  MoveL 730 to (129.65, 249.05, 0) mm, rotated rx 180 ry 0 rz -39.83 deg; joints [47.121, -60.596, 63.822, -0.862, 86.762, 47.166]
  MoveL 731 to (129.42, 249.1, 0) mm, rotated rx -180 ry 0 rz -39.83 deg; joints [47.111, -60.591, 63.814, -0.862, 86.764, 47.156]
  MoveL 732 to (129.2, 249.14, 0) mm, rotated rx -180 ry 0 rz -39.83 deg; joints [47.101, -60.586, 63.806, -0.862, 86.767, 47.146]
  MoveL 733 to (128.97, 249.18, 0) mm, rotated rx 180 ry 0 rz -39.83 deg; joints [47.091, -60.582, 63.799, -0.862, 86.769, 47.136]
  MoveL 734 to (128.75, 249.21, 0) mm, rotated rx 180 ry 0 rz -39.83 deg; joints [47.081, -60.577, 63.792, -0.862, 86.772, 47.126]
  MoveL 735 to (128.47, 249.26, 0) mm, rotated rx -180 ry 0 rz -39.83 deg; joints [47.068, -60.572, 63.784, -0.862, 86.775, 47.113]
  MoveL 736 to (128.19, 249.3, 0) mm, rotated rx 180 ry 0 rz -39.83 deg; joints [47.056, -60.567, 63.776, -0.862, 86.777, 47.101]
  MoveL 737 to (127.92, 249.33, 0) mm, rotated rx 180 ry 0 rz -39.83 deg; joints [47.043, -60.562, 63.769, -0.862, 86.78, 47.088]
  MoveL 738 to (127.64, 249.35, 0) mm, rotated rx 180 ry 0 rz -39.83 deg; joints [47.031, -60.56, 63.764, -0.862, 86.781, 47.076]
  MoveL 739 to (127.2, 249.34, 0) mm, rotated rx 180 ry 0 rz -39.83 deg; joints [47.011, -60.559, 63.762, -0.862, 86.782, 47.056]
  MoveL 740 to (126.76, 249.29, 0) mm, rotated rx 180 ry 0 rz -39.83 deg; joints [46.991, -60.561, 63.765, -0.862, 86.781, 47.036]
  MoveL 741 to (126.32, 249.21, 0) mm, rotated rx 180 ry 0 rz -39.83 deg; joints [46.97, -60.566, 63.772, -0.862, 86.779, 47.016]
  MoveL 742 to (125.88, 249.13, 0) mm, rotated rx 180 ry 0 rz -39.83 deg; joints [46.95, -60.571, 63.779, -0.862, 86.777, 46.995]
  MoveL 743 to (125.52, 249.07, 0) mm, rotated rx 180 ry 0 rz -39.83 deg; joints [46.934, -60.575, 63.784, -0.862, 86.775, 46.979]
  MoveL 744 to (125.17, 249, 0) mm, rotated rx 180 ry 0 rz -39.83 deg; joints [46.918, -60.579, 63.791, -0.862, 86.773, 46.963]
  MoveL 745 to (124.83, 248.91, 0) mm, rotated rx 180 ry 0 rz -39.83 deg; joints [46.902, -60.586, 63.8, -0.862, 86.77, 46.947]
  MoveL 746 to (124.5, 248.79, 0) mm, rotated rx 180 ry 0 rz -39.83 deg; joints [46.887, -60.595, 63.814, -0.862, 86.765, 46.932]
  MoveL 747 to (124.16, 248.61, 0) mm, rotated rx -180 ry 0 rz -39.83 deg; joints [46.871, -60.609, 63.834, -0.862, 86.759, 46.916]
  MoveL 748 to (123.85, 248.4, 0) mm, rotated rx 180 ry 0 rz -39.83 deg; joints [46.856, -60.627, 63.86, -0.862, 86.75, 46.902]
  MoveL 749 to (123.54, 248.17, 0) mm, rotated rx 180 ry 0 rz -39.83 deg; joints [46.842, -60.647, 63.89, -0.862, 86.74, 46.887]
  MoveL 750 to (123.25, 247.91, 0) mm, rotated rx 180 ry 0 rz -39.83 deg; joints [46.828, -60.668, 63.922, -0.862, 86.73, 46.874]
  MoveL 751 to (122.84, 247.54, 0) mm, rotated rx 180 ry 0 rz -39.83 deg; joints [46.808, -60.7, 63.969, -0.862, 86.714, 46.854]
  MoveL 752 to (122.44, 247.16, 0) mm, rotated rx 180 ry 0 rz -39.83 deg; joints [46.789, -60.733, 64.017, -0.862, 86.698, 46.836]
  MoveL 753 to (122.05, 246.78, 0) mm, rotated rx 180 ry 0 rz -39.83 deg; joints [46.77, -60.765, 64.065, -0.862, 86.682, 46.817]
  MoveL 754 to (121.65, 246.4, 0) mm, rotated rx 180 ry 0 rz -39.83 deg; joints [46.751, -60.797, 64.113, -0.862, 86.666, 46.798]
  MoveL 755 to (121.18, 245.95, 0) mm, rotated rx 180 ry 0 rz -39.83 deg; joints [46.728, -60.836, 64.17, -0.862, 86.648, 46.775]
  MoveL 756 to (120.69, 245.51, 0) mm, rotated rx 180 ry 0 rz -39.83 deg; joints [46.705, -60.873, 64.225, -0.862, 86.629, 46.752]
  MoveL 757 to (120.2, 245.07, 0) mm, rotated rx -180 ry 0 rz -39.83 deg; joints [46.682, -60.911, 64.28, -0.862, 86.611, 46.729]
  MoveL 758 to (119.71, 244.63, 0) mm, rotated rx 180 ry 0 rz -39.83 deg; joints [46.658, -60.948, 64.335, -0.862, 86.593, 46.706]
  MoveL 759 to (119.71, 244.63, 0) mm, rotated rx 180 ry 0 rz -39.83 deg; joints [46.658, -60.948, 64.335, -0.862, 86.593, 46.706]
  MoveL 760 to (119.52, 244.68, 0) mm, rotated rx 180 ry 0 rz -39.83 deg; joints [46.649, -60.942, 64.326, -0.862, 86.596, 46.697]
  MoveL 761 to (119.32, 244.73, 0) mm, rotated rx 180 ry 0 rz -39.83 deg; joints [46.641, -60.936, 64.318, -0.862, 86.599, 46.689]
  MoveL 762 to (119.13, 244.77, 0) mm, rotated rx 180 ry 0 rz -39.83 deg; joints [46.632, -60.932, 64.31, -0.862, 86.601, 46.68]
  MoveL 763 to (118.93, 244.79, 0) mm, rotated rx 180 ry 0 rz -39.83 deg; joints [46.623, -60.928, 64.305, -0.862, 86.603, 46.671]
  MoveL 764 to (118.67, 244.8, 0) mm, rotated rx 180 ry 0 rz -39.83 deg; joints [46.611, -60.926, 64.302, -0.862, 86.604, 46.659]
  MoveL 765 to (118.41, 244.78, 0) mm, rotated rx 180 ry 0 rz -39.83 deg; joints [46.599, -60.927, 64.303, -0.862, 86.604, 46.647]
  MoveL 766 to (118.14, 244.73, 0) mm, rotated rx 180 ry 0 rz -39.83 deg; joints [46.587, -60.929, 64.306, -0.862, 86.603, 46.635]
  MoveL 767 to (117.88, 244.68, 0) mm, rotated rx 180 ry 0 rz -39.83 deg; joints [46.575, -60.933, 64.31, -0.862, 86.602, 46.622]
  MoveL 768 to (117.41, 244.58, 0) mm, rotated rx 180 ry 0 rz -39.83 deg; joints [46.553, -60.939, 64.319, -0.862, 86.599, 46.601]
  MoveL 769 to (116.94, 244.47, 0) mm, rotated rx 180 ry 0 rz -39.83 deg; joints [46.532, -60.947, 64.33, -0.862, 86.595, 46.58]
  MoveL 770 to (116.49, 244.34, 0) mm, rotated rx 180 ry 0 rz -39.83 deg; joints [46.511, -60.956, 64.343, -0.862, 86.591, 46.558]
  MoveL 771 to (116.04, 244.18, 0) mm, rotated rx 180 ry 0 rz -39.83 deg; joints [46.49, -60.968, 64.36, -0.862, 86.585, 46.538]
  MoveL 772 to (115.64, 244.01, 0) mm, rotated rx 180 ry 0 rz -39.83 deg; joints [46.471, -60.981, 64.38, -0.862, 86.579, 46.519]
  MoveL 773 to (115.24, 243.81, 0) mm, rotated rx 180 ry 0 rz -39.83 deg; joints [46.452, -60.997, 64.403, -0.862, 86.571, 46.5]
  MoveL 774 to (114.86, 243.59, 0) mm, rotated rx 180 ry 0 rz -39.83 deg; joints [46.434, -61.014, 64.429, -0.862, 86.563, 46.482]
  MoveL 775 to (114.48, 243.35, 0) mm, rotated rx -180 ry 0 rz -39.83 deg; joints [46.417, -61.034, 64.458, -0.862, 86.553, 46.465]
  MoveL 776 to (113.98, 242.98, 0) mm, rotated rx 180 ry 0 rz -39.83 deg; joints [46.393, -61.064, 64.502, -0.862, 86.539, 46.441]
  MoveL 777 to (113.5, 242.59, 0) mm, rotated rx 180 ry 0 rz -39.83 deg; joints [46.37, -61.097, 64.551, -0.862, 86.523, 46.418]
  MoveL 778 to (113.04, 242.17, 0) mm, rotated rx 180 ry 0 rz -39.83 deg; joints [46.347, -61.132, 64.602, -0.862, 86.506, 46.396]
  MoveL 779 to (112.59, 241.74, 0) mm, rotated rx 180 ry 0 rz -39.83 deg; joints [46.326, -61.169, 64.656, -0.862, 86.488, 46.375]
  MoveL 780 to (111.99, 241.13, 0) mm, rotated rx 180 ry 0 rz -39.83 deg; joints [46.296, -61.22, 64.731, -0.862, 86.464, 46.346]
  MoveL 781 to (111.41, 240.51, 0) mm, rotated rx 180 ry 0 rz -39.83 deg; joints [46.268, -61.272, 64.809, -0.862, 86.438, 46.318]
  MoveL 782 to (110.85, 239.88, 0) mm, rotated rx 180 ry 0 rz -39.83 deg; joints [46.24, -61.326, 64.889, -0.862, 86.412, 46.291]
  MoveL 783 to (110.31, 239.22, 0) mm, rotated rx 180 ry 0 rz -39.83 deg; joints [46.214, -61.382, 64.971, -0.862, 86.385, 46.264]
  MoveL 784 to (109.76, 238.49, 0) mm, rotated rx 180 ry 0 rz -39.83 deg; joints [46.186, -61.444, 65.063, -0.862, 86.355, 46.237]
  MoveL 785 to (109.22, 237.74, 0) mm, rotated rx 180 ry 0 rz -39.83 deg; joints [46.159, -61.508, 65.157, -0.862, 86.324, 46.211]
  MoveL 786 to (108.71, 236.98, 0) mm, rotated rx 180 ry 0 rz -39.83 deg; joints [46.133, -61.573, 65.253, -0.862, 86.293, 46.185]
  MoveL 787 to (108.2, 236.22, 0) mm, rotated rx 180 ry 0 rz -39.83 deg; joints [46.107, -61.639, 65.35, -0.862, 86.261, 46.16]
  MoveL 788 to (107.72, 235.51, 0) mm, rotated rx -180 ry 0 rz -39.83 deg; joints [46.083, -61.7, 65.44, -0.862, 86.232, 46.137]
  MoveL 789 to (107.26, 234.79, 0) mm, rotated rx 180 ry 0 rz -39.83 deg; joints [46.06, -61.761, 65.531, -0.862, 86.203, 46.113]
  MoveL 790 to (106.8, 234.06, 0) mm, rotated rx 180 ry 0 rz -39.83 deg; joints [46.036, -61.823, 65.622, -0.862, 86.173, 46.09]
  MoveL 791 to (106.36, 233.33, 0) mm, rotated rx -180 ry 0 rz -39.83 deg; joints [46.014, -61.887, 65.715, -0.862, 86.143, 46.068]
  MoveL 792 to (105.88, 232.45, 0) mm, rotated rx 180 ry 0 rz -39.83 deg; joints [45.989, -61.962, 65.826, -0.862, 86.107, 46.044]
  MoveL 793 to (105.42, 231.55, 0) mm, rotated rx 180 ry 0 rz -39.83 deg; joints [45.965, -62.04, 65.94, -0.862, 86.07, 46.02]
  MoveL 794 to (104.99, 230.64, 0) mm, rotated rx 180 ry 0 rz -39.83 deg; joints [45.942, -62.118, 66.056, -0.862, 86.032, 45.998]
  MoveL 795 to (104.58, 229.72, 0) mm, rotated rx -180 ry 0 rz -39.83 deg; joints [45.92, -62.198, 66.173, -0.862, 85.995, 45.977]
  MoveL 796 to (104.2, 228.81, 0) mm, rotated rx -180 ry 0 rz -39.83 deg; joints [45.899, -62.276, 66.288, -0.862, 85.958, 45.957]
  MoveL 797 to (103.82, 227.9, 0) mm, rotated rx -180 ry 0 rz -39.83 deg; joints [45.879, -62.355, 66.403, -0.862, 85.921, 45.937]
  MoveL 798 to (103.46, 226.99, 0) mm, rotated rx -180 ry 0 rz -39.83 deg; joints [45.859, -62.434, 66.519, -0.862, 85.884, 45.917]
  MoveL 799 to (103.09, 226.08, 0) mm, rotated rx 180 ry 0 rz -39.83 deg; joints [45.839, -62.513, 66.634, -0.862, 85.847, 45.898]
  MoveL 800 to (102.74, 225.23, 0) mm, rotated rx -180 ry 0 rz -39.83 deg; joints [45.82, -62.586, 66.741, -0.862, 85.812, 45.879]
  MoveL 801 to (102.4, 224.39, 0) mm, rotated rx 180 ry 0 rz -39.83 deg; joints [45.801, -62.658, 66.848, -0.862, 85.779, 45.861]
  MoveL 802 to (102.05, 223.54, 0) mm, rotated rx 180 ry 0 rz -39.83 deg; joints [45.782, -62.731, 66.954, -0.862, 85.745, 45.842]
  MoveL 803 to (101.69, 222.7, 0) mm, rotated rx 180 ry 0 rz -39.83 deg; joints [45.762, -62.803, 67.059, -0.862, 85.711, 45.823]
  MoveL 804 to (101.69, 222.7, 0) mm, rotated rx 180 ry 0 rz -39.83 deg; joints [45.762, -62.803, 67.059, -0.862, 85.711, 45.823]
  MoveL 805 to (101.34, 223.54, 0) mm, rotated rx 180 ry 0 rz -39.83 deg; joints [45.749, -62.726, 66.946, -0.862, 85.747, 45.81]
  MoveL 806 to (100.99, 224.39, 0) mm, rotated rx -180 ry 0 rz -39.83 deg; joints [45.736, -62.649, 66.832, -0.862, 85.784, 45.796]
  MoveL 807 to (100.64, 225.23, 0) mm, rotated rx 180 ry 0 rz -39.83 deg; joints [45.723, -62.572, 66.718, -0.862, 85.82, 45.782]
  MoveL 808 to (100.3, 226.08, 0) mm, rotated rx 180 ry 0 rz -39.83 deg; joints [45.71, -62.494, 66.603, -0.862, 85.857, 45.769]
  MoveL 809 to (99.93, 226.99, 0) mm, rotated rx -180 ry 0 rz -39.83 deg; joints [45.696, -62.41, 66.48, -0.862, 85.897, 45.755]
  MoveL 810 to (99.56, 227.9, 0) mm, rotated rx 180 ry 0 rz -39.83 deg; joints [45.683, -62.327, 66.356, -0.862, 85.937, 45.74]
  MoveL 811 to (99.19, 228.81, 0) mm, rotated rx 180 ry 0 rz -39.83 deg; joints [45.669, -62.243, 66.232, -0.862, 85.977, 45.726]
  MoveL 812 to (98.81, 229.72, 0) mm, rotated rx -180 ry 0 rz -39.83 deg; joints [45.655, -62.159, 66.108, -0.862, 86.017, 45.711]
  MoveL 813 to (98.4, 230.64, 0) mm, rotated rx 180 ry 0 rz -39.83 deg; joints [45.639, -62.074, 65.982, -0.862, 86.058, 45.695]
  MoveL 814 to (97.97, 231.55, 0) mm, rotated rx 180 ry 0 rz -39.83 deg; joints [45.623, -61.99, 65.857, -0.862, 86.098, 45.678]
  MoveL 815 to (97.51, 232.45, 0) mm, rotated rx 180 ry 0 rz -39.83 deg; joints [45.605, -61.906, 65.733, -0.862, 86.139, 45.66]
  MoveL 816 to (97.03, 233.33, 0) mm, rotated rx 180 ry 0 rz -39.83 deg; joints [45.586, -61.824, 65.61, -0.862, 86.178, 45.64]
  MoveL 817 to (96.59, 234.06, 0) mm, rotated rx 180 ry 0 rz -39.83 deg; joints [45.569, -61.755, 65.507, -0.862, 86.212, 45.622]
  MoveL 818 to (96.13, 234.79, 0) mm, rotated rx 180 ry 0 rz -39.83 deg; joints [45.551, -61.687, 65.406, -0.862, 86.245, 45.604]
  MoveL 819 to (95.67, 235.51, 0) mm, rotated rx -180 ry 0 rz -39.83 deg; joints [45.532, -61.619, 65.305, -0.862, 86.278, 45.584]
  MoveL 820 to (95.19, 236.22, 0) mm, rotated rx 180 ry 0 rz -39.83 deg; joints [45.513, -61.552, 65.204, -0.862, 86.311, 45.565]
  MoveL 821 to (94.68, 236.98, 0) mm, rotated rx 180 ry 0 rz -39.83 deg; joints [45.493, -61.479, 65.096, -0.862, 86.347, 45.544]
  MoveL 822 to (94.16, 237.74, 0) mm, rotated rx 180 ry 0 rz -39.83 deg; joints [45.472, -61.407, 64.988, -0.862, 86.382, 45.523]
  MoveL 823 to (93.63, 238.49, 0) mm, rotated rx -180 ry 0 rz -39.83 deg; joints [45.45, -61.336, 64.881, -0.861, 86.417, 45.501]
  MoveL 824 to (93.08, 239.22, 0) mm, rotated rx 180 ry 0 rz -39.83 deg; joints [45.428, -61.266, 64.777, -0.861, 86.452, 45.478]
  MoveL 825 to (92.54, 239.88, 0) mm, rotated rx 180 ry 0 rz -39.83 deg; joints [45.406, -61.203, 64.682, -0.861, 86.483, 45.455]
  MoveL 826 to (91.98, 240.51, 0) mm, rotated rx 180 ry 0 rz -39.83 deg; joints [45.383, -61.142, 64.589, -0.861, 86.514, 45.432]
  MoveL 827 to (91.39, 241.13, 0) mm, rotated rx 180 ry 0 rz -39.83 deg; joints [45.359, -61.081, 64.498, -0.861, 86.544, 45.407]
  MoveL 828 to (90.79, 241.74, 0) mm, rotated rx 180 ry 0 rz -39.83 deg; joints [45.334, -61.022, 64.409, -0.861, 86.574, 45.382]
  MoveL 829 to (90.35, 242.17, 0) mm, rotated rx 180 ry 0 rz -39.83 deg; joints [45.315, -60.98, 64.346, -0.861, 86.595, 45.362]
  MoveL 830 to (89.88, 242.59, 0) mm, rotated rx -180 ry 0 rz -39.83 deg; joints [45.295, -60.939, 64.283, -0.861, 86.615, 45.343]
  MoveL 831 to (89.4, 242.98, 0) mm, rotated rx 180 ry 0 rz -39.83 deg; joints [45.275, -60.899, 64.224, -0.861, 86.635, 45.322]
  MoveL 832 to (88.9, 243.35, 0) mm, rotated rx 180 ry 0 rz -39.83 deg; joints [45.254, -60.862, 64.168, -0.861, 86.654, 45.301]
  MoveL 833 to (88.53, 243.59, 0) mm, rotated rx 180 ry 0 rz -39.83 deg; joints [45.238, -60.837, 64.13, -0.861, 86.667, 45.285]
  MoveL 834 to (88.15, 243.81, 0) mm, rotated rx 180 ry 0 rz -39.83 deg; joints [45.221, -60.815, 64.095, -0.861, 86.678, 45.268]
  MoveL 835 to (87.75, 244.01, 0) mm, rotated rx 180 ry 0 rz -39.83 deg; joints [45.204, -60.793, 64.063, -0.861, 86.689, 45.251]
  MoveL 836 to (87.35, 244.18, 0) mm, rotated rx 180 ry 0 rz -39.83 deg; joints [45.187, -60.775, 64.035, -0.861, 86.698, 45.233]
  MoveL 837 to (86.9, 244.34, 0) mm, rotated rx 180 ry 0 rz -39.83 deg; joints [45.167, -60.757, 64.008, -0.861, 86.708, 45.213]
  MoveL 838 to (86.44, 244.47, 0) mm, rotated rx 180 ry 0 rz -39.83 deg; joints [45.147, -60.742, 63.984, -0.861, 86.716, 45.193]
  MoveL 839 to (85.98, 244.58, 0) mm, rotated rx 180 ry 0 rz -39.83 deg; joints [45.126, -60.728, 63.963, -0.861, 86.723, 45.172]
  MoveL 840 to (85.51, 244.68, 0) mm, rotated rx 180 ry 0 rz -39.83 deg; joints [45.105, -60.715, 63.943, -0.861, 86.729, 45.151]
  MoveL 841 to (85.25, 244.73, 0) mm, rotated rx 180 ry 0 rz -39.83 deg; joints [45.094, -60.708, 63.932, -0.861, 86.733, 45.139]
  MoveL 842 to (84.98, 244.78, 0) mm, rotated rx 180 ry 0 rz -39.83 deg; joints [45.082, -60.702, 63.923, -0.861, 86.736, 45.127]
  MoveL 843 to (84.72, 244.8, 0) mm, rotated rx 180 ry 0 rz -39.83 deg; joints [45.07, -60.698, 63.917, -0.861, 86.738, 45.115]
  MoveL 844 to (84.45, 244.79, 0) mm, rotated rx 180 ry 0 rz -39.83 deg; joints [45.058, -60.696, 63.914, -0.861, 86.739, 45.103]
  MoveL 845 to (84.26, 244.77, 0) mm, rotated rx 180 ry 0 rz -39.83 deg; joints [45.049, -60.697, 63.915, -0.861, 86.739, 45.094]
  MoveL 846 to (84.06, 244.73, 0) mm, rotated rx 180 ry 0 rz -39.83 deg; joints [45.04, -60.699, 63.917, -0.861, 86.738, 45.085]
  MoveL 847 to (83.87, 244.68, 0) mm, rotated rx 180 ry 0 rz -39.83 deg; joints [45.031, -60.702, 63.921, -0.861, 86.737, 45.077]
  MoveL 848 to (83.68, 244.63, 0) mm, rotated rx 180 ry 0 rz -39.83 deg; joints [45.022, -60.705, 63.926, -0.861, 86.735, 45.068]
  Establecer velocidad (1000.0 mm/s)
  MoveL 849 to (83.68, 244.63, 0) mm, rotated rx 180 ry 0 rz -39.83 deg; joints [45.022, -60.705, 63.926, -0.861, 86.735, 45.068]
  MoveL 850 to (83.68, 244.63, 20) mm, rotated rx 180 ry 0 rz -39.83 deg; joints [45.036, -60.88, 62.472, -0.86, 88.364, 45.057]

--- program P_ou_2 (robot KUKA KR 16 2) ---
  Suave(1)
  Establecer velocidad (1000.0 mm/s)
  Est. Ref.: Frame 2
  Est. herr: Plumon_ensamble
  Mostrar Plumon_ensamble
  MoveJ 1 to (72.95, 248.83, 20) mm, rotated rx 180 ry 0 rz -39.83 deg; joints [44.569, -60.401, 61.74, -0.859, 88.61, 44.586]
  MoveL 2 to (72.95, 248.83, 20) mm, rotated rx 180 ry 0 rz -39.83 deg; joints [44.569, -60.401, 61.74, -0.859, 88.61, 44.586]
  MoveL 3 to (72.95, 248.83, 0) mm, rotated rx 180 ry 0 rz -39.83 deg; joints [44.555, -60.233, 63.202, -0.86, 86.979, 44.597]
  MoveL 4 to (72.95, 248.83, 0) mm, rotated rx 180 ry 0 rz -39.83 deg; joints [44.555, -60.233, 63.202, -0.86, 86.979, 44.597]
  Establecer velocidad (50.0 mm/s)
  MoveL 5 to (73.14, 248.89, 0) mm, rotated rx -180 ry 0 rz -39.83 deg; joints [44.564, -60.229, 63.197, -0.86, 86.981, 44.606]
  MoveL 6 to (73.34, 248.95, 0) mm, rotated rx 180 ry 0 rz -39.83 deg; joints [44.574, -60.226, 63.192, -0.86, 86.983, 44.615]
  MoveL 7 to (73.54, 249, 0) mm, rotated rx 180 ry 0 rz -39.83 deg; joints [44.583, -60.223, 63.188, -0.86, 86.984, 44.624]
  MoveL 8 to (73.74, 249.05, 0) mm, rotated rx -180 ry 0 rz -39.83 deg; joints [44.592, -60.22, 63.184, -0.86, 86.985, 44.634]
  MoveL 9 to (73.96, 249.1, 0) mm, rotated rx 180 ry 0 rz -39.83 deg; joints [44.602, -60.218, 63.181, -0.86, 86.986, 44.644]
  MoveL 10 to (74.19, 249.14, 0) mm, rotated rx 180 ry 0 rz -39.83 deg; joints [44.613, -60.216, 63.178, -0.86, 86.987, 44.654]
  MoveL 11 to (74.41, 249.18, 0) mm, rotated rx -180 ry 0 rz -39.83 deg; joints [44.623, -60.214, 63.176, -0.86, 86.988, 44.664]
  MoveL 12 to (74.64, 249.21, 0) mm, rotated rx 180 ry 0 rz -39.83 deg; joints [44.633, -60.213, 63.175, -0.86, 86.988, 44.675]
  MoveL 13 to (74.92, 249.26, 0) mm, rotated rx 180 ry 0 rz -39.83 deg; joints [44.646, -60.211, 63.172, -0.86, 86.989, 44.688]
  MoveL 14 to (75.19, 249.3, 0) mm, rotated rx 180 ry 0 rz -39.83 deg; joints [44.659, -60.21, 63.171, -0.86, 86.99, 44.7]
  MoveL 15 to (75.47, 249.33, 0) mm, rotated rx 180 ry 0 rz -39.83 deg; joints [44.671, -60.209, 63.17, -0.86, 86.99, 44.713]
  MoveL 16 to (75.75, 249.35, 0) mm, rotated rx 180 ry 0 rz -39.83 deg; joints [44.684, -60.21, 63.172, -0.86, 86.989, 44.725]
  MoveL 17 to (76.19, 249.34, 0) mm, rotated rx 180 ry 0 rz -39.83 deg; joints [44.703, -60.215, 63.18, -0.86, 86.986, 44.745]
  MoveL 18 to (76.63, 249.29, 0) mm, rotated rx 180 ry 0 rz -39.83 deg; joints [44.723, -60.223, 63.193, -0.86, 86.982, 44.765]
  MoveL 19 to (77.07, 249.21, 0) mm, rotated rx 180 ry 0 rz -39.83 deg; joints [44.743, -60.234, 63.209, -0.86, 86.976, 44.784]
  MoveL 20 to (77.51, 249.13, 0) mm, rotated rx 180 ry 0 rz -39.83 deg; joints [44.762, -60.245, 63.227, -0.86, 86.97, 44.804]
  MoveL 21 to (77.87, 249.07, 0) mm, rotated rx 180 ry 0 rz -39.83 deg; joints [44.778, -60.254, 63.24, -0.86, 86.966, 44.82]
  MoveL 22 to (78.22, 249, 0) mm, rotated rx 180 ry 0 rz -39.83 deg; joints [44.794, -60.263, 63.255, -0.861, 86.961, 44.836]
  MoveL 23 to (78.56, 248.91, 0) mm, rotated rx 180 ry 0 rz -39.83 deg; joints [44.809, -60.274, 63.272, -0.861, 86.955, 44.851]
  MoveL 24 to (78.89, 248.79, 0) mm, rotated rx 180 ry 0 rz -39.83 deg; joints [44.823, -60.288, 63.293, -0.861, 86.948, 44.865]
  MoveL 25 to (79.23, 248.61, 0) mm, rotated rx 180 ry 0 rz -39.83 deg; joints [44.837, -60.307, 63.322, -0.861, 86.938, 44.88]
  MoveL 26 to (79.54, 248.4, 0) mm, rotated rx 180 ry 0 rz -39.83 deg; joints [44.851, -60.328, 63.355, -0.861, 86.927, 44.893]
  MoveL 27 to (79.84, 248.17, 0) mm, rotated rx 180 ry 0 rz -39.83 deg; joints [44.863, -60.353, 63.392, -0.861, 86.915, 44.906]
  MoveL 28 to (80.14, 247.91, 0) mm, rotated rx 180 ry 0 rz -39.83 deg; joints [44.876, -60.378, 63.43, -0.861, 86.902, 44.918]
  MoveL 29 to (80.54, 247.54, 0) mm, rotated rx -180 ry 0 rz -39.83 deg; joints [44.892, -60.415, 63.487, -0.861, 86.882, 44.936]
  MoveL 30 to (80.94, 247.16, 0) mm, rotated rx 180 ry 0 rz -39.83 deg; joints [44.909, -60.453, 63.544, -0.861, 86.863, 44.952]
  MoveL 31 to (81.34, 246.78, 0) mm, rotated rx 180 ry 0 rz -39.83 deg; joints [44.925, -60.491, 63.602, -0.861, 86.844, 44.969]
  MoveL 32 to (81.73, 246.4, 0) mm, rotated rx 180 ry 0 rz -39.83 deg; joints [44.941, -60.529, 63.659, -0.861, 86.825, 44.986]
  MoveL 33 to (82.21, 245.95, 0) mm, rotated rx 180 ry 0 rz -39.83 deg; joints [44.961, -60.574, 63.726, -0.861, 86.802, 45.006]
  MoveL 34 to (82.7, 245.51, 0) mm, rotated rx 180 ry 0 rz -39.83 deg; joints [44.981, -60.618, 63.793, -0.861, 86.78, 45.026]
  MoveL 35 to (83.18, 245.07, 0) mm, rotated rx 180 ry 0 rz -39.83 deg; joints [45.002, -60.662, 63.86, -0.861, 86.757, 45.047]
  MoveL 36 to (83.68, 244.63, 0) mm, rotated rx 180 ry 0 rz -39.83 deg; joints [45.022, -60.705, 63.926, -0.861, 86.735, 45.068]
  Establecer velocidad (1000.0 mm/s)
  MoveL 37 to (83.68, 244.63, 0) mm, rotated rx 180 ry 0 rz -39.83 deg; joints [45.022, -60.705, 63.926, -0.861, 86.735, 45.068]
  MoveL 38 to (83.68, 244.63, 20) mm, rotated rx 180 ry 0 rz -39.83 deg; joints [45.036, -60.88, 62.472, -0.86, 88.364, 45.057]
  Establecer velocidad (1000.0 mm/s)
  MoveL 39 to (72.95, 248.83, 20) mm, rotated rx 180 ry 0 rz -39.83 deg; joints [44.569, -60.401, 61.74, -0.859, 88.61, 44.586]
  MoveL 40 to (72.95, 248.83, 0) mm, rotated rx 180 ry 0 rz -39.83 deg; joints [44.555, -60.233, 63.202, -0.86, 86.979, 44.597]
  MoveL 41 to (72.95, 248.83, 0) mm, rotated rx 180 ry 0 rz -39.83 deg; joints [44.555, -60.233, 63.202, -0.86, 86.979, 44.597]
  Establecer velocidad (50.0 mm/s)
  MoveL 42 to (72.46, 249.17, 0) mm, rotated rx 180 ry 0 rz -39.83 deg; joints [44.535, -60.197, 63.148, -0.86, 86.998, 44.576]
  MoveL 43 to (71.96, 249.51, 0) mm, rotated rx 180 ry 0 rz -39.83 deg; joints [44.514, -60.163, 63.095, -0.86, 87.015, 44.555]
  MoveL 44 to (71.46, 249.82, 0) mm, rotated rx 180 ry 0 rz -39.83 deg; joints [44.493, -60.129, 63.044, -0.86, 87.033, 44.534]
  MoveL 45 to (70.94, 250.12, 0) mm, rotated rx 180 ry 0 rz -39.83 deg; joints [44.471, -60.097, 62.996, -0.86, 87.049, 44.511]
  MoveL 46 to (70.56, 250.31, 0) mm, rotated rx -180 ry 0 rz -39.83 deg; joints [44.454, -60.076, 62.963, -0.86, 87.06, 44.495]
  MoveL 47 to (70.17, 250.49, 0) mm, rotated rx 180 ry 0 rz -39.83 deg; joints [44.438, -60.057, 62.933, -0.86, 87.07, 44.478]
  MoveL 48 to (69.78, 250.65, 0) mm, rotated rx 180 ry 0 rz -39.83 deg; joints [44.421, -60.039, 62.906, -0.86, 87.08, 44.461]
  MoveL 49 to (69.37, 250.78, 0) mm, rotated rx 180 ry 0 rz -39.83 deg; joints [44.403, -60.023, 62.882, -0.86, 87.088, 44.443]
  MoveL 50 to (69.02, 250.87, 0) mm, rotated rx 180 ry 0 rz -39.83 deg; joints [44.387, -60.012, 62.864, -0.86, 87.094, 44.427]
  MoveL 51 to (68.66, 250.94, 0) mm, rotated rx 180 ry 0 rz -39.83 deg; joints [44.372, -60.002, 62.849, -0.86, 87.099, 44.412]
  MoveL 52 to (68.31, 251, 0) mm, rotated rx 180 ry 0 rz -39.83 deg; joints [44.356, -59.993, 62.835, -0.86, 87.104, 44.396]
  MoveL 53 to (67.95, 251.04, 0) mm, rotated rx 180 ry 0 rz -39.83 deg; joints [44.34, -59.986, 62.824, -0.86, 87.108, 44.38]
  MoveL 54 to (67.64, 251.06, 0) mm, rotated rx 180 ry 0 rz -39.83 deg; joints [44.326, -59.981, 62.816, -0.86, 87.11, 44.366]
  MoveL 55 to (67.33, 251.08, 0) mm, rotated rx 180 ry 0 rz -39.83 deg; joints [44.313, -59.977, 62.81, -0.86, 87.113, 44.352]
  MoveL 56 to (67.03, 251.08, 0) mm, rotated rx 180 ry 0 rz -39.83 deg; joints [44.299, -59.974, 62.805, -0.86, 87.114, 44.339]
  MoveL 57 to (66.72, 251.06, 0) mm, rotated rx -180 ry 0 rz -39.83 deg; joints [44.285, -59.973, 62.802, -0.86, 87.115, 44.325]
  MoveL 58 to (66.4, 251.03, 0) mm, rotated rx 180 ry 0 rz -39.83 deg; joints [44.271, -59.973, 62.802, -0.86, 87.115, 44.31]
  MoveL 59 to (66.09, 250.98, 0) mm, rotated rx 180 ry 0 rz -39.83 deg; joints [44.256, -59.974, 62.804, -0.86, 87.115, 44.296]
  MoveL 60 to (65.78, 250.91, 0) mm, rotated rx 180 ry 0 rz -39.83 deg; joints [44.242, -59.978, 62.809, -0.86, 87.113, 44.282]
  MoveL 61 to (65.47, 250.82, 0) mm, rotated rx 180 ry 0 rz -39.83 deg; joints [44.228, -59.983, 62.816, -0.86, 87.111, 44.268]
  MoveL 62 to (65.14, 250.7, 0) mm, rotated rx 180 ry 0 rz -39.83 deg; joints [44.212, -59.991, 62.828, -0.86, 87.107, 44.252]
  MoveL 63 to (64.81, 250.56, 0) mm, rotated rx 180 ry 0 rz -39.83 deg; joints [44.197, -60.001, 62.842, -0.86, 87.102, 44.237]
  MoveL 64 to (64.48, 250.41, 0) mm, rotated rx 180 ry 0 rz -39.83 deg; joints [44.181, -60.011, 62.858, -0.86, 87.097, 44.221]
  MoveL 65 to (64.16, 250.25, 0) mm, rotated rx 180 ry 0 rz -39.83 deg; joints [44.166, -60.023, 62.874, -0.86, 87.091, 44.206]
  MoveL 66 to (64.16, 250.25, 0) mm, rotated rx 180 ry 0 rz -39.83 deg; joints [44.166, -60.023, 62.874, -0.86, 87.091, 44.206]
  MoveL 67 to (63.61, 250.48, 0) mm, rotated rx 180 ry 0 rz -39.83 deg; joints [44.143, -59.996, 62.834, -0.86, 87.105, 44.182]
  MoveL 68 to (63.06, 250.71, 0) mm, rotated rx 180 ry 0 rz -39.83 deg; joints [44.119, -59.97, 62.794, -0.86, 87.119, 44.159]
  MoveL 69 to (62.51, 250.94, 0) mm, rotated rx 180 ry 0 rz -39.83 deg; joints [44.095, -59.944, 62.753, -0.86, 87.133, 44.135]
  MoveL 70 to (61.96, 251.17, 0) mm, rotated rx -180 ry 0 rz -39.83 deg; joints [44.072, -59.918, 62.713, -0.86, 87.146, 44.111]
  MoveL 71 to (61.51, 251.36, 0) mm, rotated rx 180 ry 0 rz -39.83 deg; joints [44.052, -59.896, 62.68, -0.86, 87.157, 44.091]
  MoveL 72 to (61.05, 251.54, 0) mm, rotated rx -180 ry 0 rz -39.83 deg; joints [44.033, -59.875, 62.648, -0.86, 87.168, 44.071]
  MoveL 73 to (60.59, 251.7, 0) mm, rotated rx 180 ry 0 rz -39.83 deg; joints [44.013, -59.856, 62.618, -0.86, 87.179, 44.051]
  MoveL 74 to (60.12, 251.85, 0) mm, rotated rx 180 ry 0 rz -39.83 deg; joints [43.993, -59.838, 62.59, -0.86, 87.188, 44.031]
  MoveL 75 to (59.67, 251.97, 0) mm, rotated rx 180 ry 0 rz -39.83 deg; joints [43.973, -59.822, 62.566, -0.86, 87.196, 44.011]
  MoveL 76 to (59.2, 252.07, 0) mm, rotated rx 180 ry 0 rz -39.83 deg; joints [43.952, -59.808, 62.544, -0.86, 87.204, 43.991]
  MoveL 77 to (58.74, 252.15, 0) mm, rotated rx 180 ry 0 rz -39.83 deg; joints [43.932, -59.796, 62.525, -0.86, 87.21, 43.97]
  MoveL 78 to (58.26, 252.22, 0) mm, rotated rx 180 ry 0 rz -39.83 deg; joints [43.911, -59.785, 62.508, -0.859, 87.216, 43.949]
  MoveL 79 to (57.81, 252.27, 0) mm, rotated rx 180 ry 0 rz -39.83 deg; joints [43.891, -59.776, 62.494, -0.859, 87.221, 43.929]
  MoveL 80 to (57.35, 252.3, 0) mm, rotated rx 180 ry 0 rz -39.83 deg; joints [43.87, -59.769, 62.482, -0.859, 87.225, 43.908]
  MoveL 81 to (56.9, 252.3, 0) mm, rotated rx -180 ry 0 rz -39.83 deg; joints [43.85, -59.765, 62.476, -0.859, 87.228, 43.888]
  MoveL 82 to (56.45, 252.24, 0) mm, rotated rx 180 ry 0 rz -39.83 deg; joints [43.83, -59.765, 62.476, -0.859, 87.228, 43.867]
  MoveL 83 to (56.15, 252.18, 0) mm, rotated rx 180 ry 0 rz -39.83 deg; joints [43.816, -59.768, 62.48, -0.859, 87.226, 43.854]
  MoveL 84 to (55.85, 252.09, 0) mm, rotated rx 180 ry 0 rz -39.83 deg; joints [43.802, -59.774, 62.488, -0.859, 87.224, 43.84]
  MoveL 85 to (55.56, 251.97, 0) mm, rotated rx -180 ry 0 rz -39.83 deg; joints [43.788, -59.781, 62.499, -0.859, 87.22, 43.826]
  MoveL 86 to (55.29, 251.83, 0) mm, rotated rx -180 ry 0 rz -39.83 deg; joints [43.775, -59.792, 62.514, -0.859, 87.215, 43.814]
  MoveL 87 to (54.94, 251.61, 0) mm, rotated rx 180 ry 0 rz -39.83 deg; joints [43.759, -59.808, 62.539, -0.859, 87.206, 43.797]
  MoveL 88 to (54.61, 251.35, 0) mm, rotated rx 180 ry 0 rz -39.83 deg; joints [43.743, -59.828, 62.568, -0.859, 87.197, 43.781]
  MoveL 89 to (54.3, 251.08, 0) mm, rotated rx 180 ry 0 rz -39.83 deg; joints [43.727, -59.85, 62.601, -0.859, 87.186, 43.766]
  MoveL 90 to (54, 250.8, 0) mm, rotated rx 180 ry 0 rz -39.83 deg; joints [43.712, -59.872, 62.635, -0.859, 87.174, 43.751]
  MoveL 91 to (54, 250.8, 0) mm, rotated rx 180 ry 0 rz -39.83 deg; joints [43.712, -59.872, 62.635, -0.859, 87.174, 43.751]
  MoveL 92 to (53.43, 250.97, 0) mm, rotated rx 180 ry 0 rz -39.83 deg; joints [43.688, -59.851, 62.602, -0.859, 87.185, 43.726]
  MoveL 93 to (52.87, 251.14, 0) mm, rotated rx 180 ry 0 rz -39.83 deg; joints [43.664, -59.83, 62.569, -0.859, 87.196, 43.702]
  MoveL 94 to (52.31, 251.3, 0) mm, rotated rx 180 ry 0 rz -39.83 deg; joints [43.639, -59.809, 62.537, -0.859, 87.208, 43.677]
  MoveL 95 to (51.75, 251.46, 0) mm, rotated rx 180 ry 0 rz -39.83 deg; joints [43.615, -59.789, 62.505, -0.859, 87.218, 43.653]
  MoveL 96 to (51.24, 251.6, 0) mm, rotated rx 180 ry 0 rz -39.83 deg; joints [43.593, -59.77, 62.477, -0.859, 87.228, 43.631]
  MoveL 97 to (50.73, 251.74, 0) mm, rotated rx 180 ry 0 rz -39.83 deg; joints [43.571, -59.753, 62.449, -0.859, 87.238, 43.608]
  MoveL 98 to (50.22, 251.86, 0) mm, rotated rx 180 ry 0 rz -39.83 deg; joints [43.548, -59.736, 62.424, -0.859, 87.246, 43.586]
  MoveL 99 to (49.7, 251.97, 0) mm, rotated rx 180 ry 0 rz -39.83 deg; joints [43.526, -59.721, 62.4, -0.859, 87.255, 43.563]
  MoveL 100 to (49.24, 252.04, 0) mm, rotated rx 180 ry 0 rz -39.83 deg; joints [43.506, -59.709, 62.381, -0.859, 87.261, 43.543]
  MoveL 101 to (48.78, 252.09, 0) mm, rotated rx -180 ry 0 rz -39.83 deg; joints [43.485, -59.7, 62.366, -0.859, 87.266, 43.522]
  MoveL 102 to (48.31, 252.11, 0) mm, rotated rx 180 ry 0 rz -39.83 deg; joints [43.464, -59.693, 62.356, -0.859, 87.27, 43.502]
  MoveL 103 to (47.85, 252.08, 0) mm, rotated rx 180 ry 0 rz -39.83 deg; joints [43.444, -59.691, 62.353, -0.859, 87.271, 43.481]
  MoveL 104 to (47.49, 252.02, 0) mm, rotated rx 180 ry 0 rz -39.83 deg; joints [43.427, -59.693, 62.355, -0.859, 87.27, 43.464]
  MoveL 105 to (47.13, 251.93, 0) mm, rotated rx 180 ry 0 rz -39.83 deg; joints [43.411, -59.697, 62.361, -0.859, 87.268, 43.448]
  MoveL 106 to (46.78, 251.82, 0) mm, rotated rx 180 ry 0 rz -39.83 deg; joints [43.394, -59.703, 62.37, -0.859, 87.265, 43.431]
  MoveL 107 to (46.42, 251.7, 0) mm, rotated rx 180 ry 0 rz -39.83 deg; joints [43.378, -59.71, 62.379, -0.859, 87.262, 43.415]
  MoveL 108 to (46.04, 251.58, 0) mm, rotated rx 180 ry 0 rz -39.83 deg; joints [43.36, -59.718, 62.391, -0.859, 87.258, 43.397]
  MoveL 109 to (45.67, 251.44, 0) mm, rotated rx 180 ry 0 rz -39.83 deg; joints [43.342, -59.727, 62.403, -0.859, 87.254, 43.38]
  MoveL 110 to (45.3, 251.28, 0) mm, rotated rx 180 ry 0 rz -39.83 deg; joints [43.325, -59.737, 62.419, -0.859, 87.249, 43.363]
  MoveL 111 to (44.95, 251.09, 0) mm, rotated rx 180 ry 0 rz -39.83 deg; joints [43.308, -59.751, 62.439, -0.859, 87.242, 43.346]
  MoveL 112 to (44.71, 250.93, 0) mm, rotated rx -180 ry 0 rz -39.83 deg; joints [43.297, -59.762, 62.456, -0.859, 87.236, 43.335]
  MoveL 113 to (44.49, 250.76, 0) mm, rotated rx 180 ry 0 rz -39.83 deg; joints [43.286, -59.776, 62.476, -0.859, 87.23, 43.324]
  MoveL 114 to (44.28, 250.57, 0) mm, rotated rx 180 ry 0 rz -39.83 deg; joints [43.276, -59.791, 62.498, -0.859, 87.222, 43.314]
  MoveL 115 to (44.09, 250.36, 0) mm, rotated rx 180 ry 0 rz -39.83 deg; joints [43.266, -59.808, 62.524, -0.859, 87.214, 43.304]
  MoveL 116 to (43.99, 250.23, 0) mm, rotated rx 180 ry 0 rz -39.83 deg; joints [43.261, -59.819, 62.54, -0.859, 87.208, 43.299]
  MoveL 117 to (43.89, 250.09, 0) mm, rotated rx 180 ry 0 rz -39.83 deg; joints [43.255, -59.83, 62.557, -0.859, 87.202, 43.294]
  MoveL 118 to (43.79, 249.96, 0) mm, rotated rx 180 ry 0 rz -39.83 deg; joints [43.25, -59.842, 62.575, -0.859, 87.196, 43.289]
  MoveL 119 to (43.7, 249.81, 0) mm, rotated rx 180 ry 0 rz -39.83 deg; joints [43.245, -59.853, 62.593, -0.859, 87.19, 43.284]
  MoveL 120 to (43.7, 249.81, 0) mm, rotated rx 180 ry 0 rz -39.83 deg; joints [43.245, -59.853, 62.593, -0.859, 87.19, 43.284]
  MoveL 121 to (43.28, 249.87, 0) mm, rotated rx 180 ry 0 rz -39.83 deg; joints [43.227, -59.844, 62.577, -0.859, 87.196, 43.265]
  MoveL 122 to (42.86, 249.93, 0) mm, rotated rx -180 ry 0 rz -39.83 deg; joints [43.208, -59.834, 62.562, -0.859, 87.201, 43.247]
  MoveL 123 to (42.44, 249.97, 0) mm, rotated rx 180 ry 0 rz -39.83 deg; joints [43.19, -59.825, 62.548, -0.859, 87.206, 43.228]
  MoveL 124 to (42.02, 250.01, 0) mm, rotated rx 180 ry 0 rz -39.83 deg; joints [43.171, -59.817, 62.535, -0.859, 87.21, 43.209]
  MoveL 125 to (41.49, 250.04, 0) mm, rotated rx 180 ry 0 rz -39.83 deg; joints [43.148, -59.809, 62.522, -0.859, 87.214, 43.186]
  MoveL 126 to (40.96, 250.04, 0) mm, rotated rx 180 ry 0 rz -39.83 deg; joints [43.124, -59.803, 62.512, -0.859, 87.218, 43.162]
  MoveL 127 to (40.43, 250.01, 0) mm, rotated rx 180 ry 0 rz -39.83 deg; joints [43.1, -59.8, 62.507, -0.859, 87.22, 43.138]
  MoveL 128 to (39.91, 249.94, 0) mm, rotated rx 180 ry 0 rz -39.83 deg; joints [43.076, -59.8, 62.506, -0.858, 87.22, 43.114]
  MoveL 129 to (39.54, 249.88, 0) mm, rotated rx -180 ry 0 rz -39.83 deg; joints [43.059, -59.802, 62.509, -0.858, 87.219, 43.097]
  MoveL 130 to (39.17, 249.79, 0) mm, rotated rx -180 ry 0 rz -39.83 deg; joints [43.042, -59.805, 62.514, -0.858, 87.218, 43.08]
  MoveL 131 to (38.8, 249.7, 0) mm, rotated rx 180 ry 0 rz -39.83 deg; joints [43.025, -59.81, 62.52, -0.858, 87.216, 43.063]
  MoveL 132 to (38.43, 249.59, 0) mm, rotated rx 180 ry 0 rz -39.83 deg; joints [43.008, -59.815, 62.528, -0.858, 87.213, 43.046]
  MoveL 133 to (38.16, 249.51, 0) mm, rotated rx -180 ry 0 rz -39.83 deg; joints [42.995, -59.819, 62.534, -0.858, 87.211, 43.033]
  MoveL 134 to (37.88, 249.42, 0) mm, rotated rx 180 ry 0 rz -39.83 deg; joints [42.983, -59.824, 62.541, -0.858, 87.209, 43.021]
  MoveL 135 to (37.61, 249.32, 0) mm, rotated rx 180 ry 0 rz -39.83 deg; joints [42.97, -59.831, 62.55, -0.858, 87.206, 43.008]
  MoveL 136 to (37.36, 249.2, 0) mm, rotated rx 180 ry 0 rz -39.83 deg; joints [42.958, -59.839, 62.562, -0.858, 87.202, 42.996]
  MoveL 137 to (37.13, 249.06, 0) mm, rotated rx 180 ry 0 rz -39.83 deg; joints [42.947, -59.849, 62.577, -0.858, 87.197, 42.985]
  MoveL 138 to (36.91, 248.91, 0) mm, rotated rx 180 ry 0 rz -39.83 deg; joints [42.936, -59.86, 62.594, -0.858, 87.191, 42.975]
  MoveL 139 to (36.7, 248.74, 0) mm, rotated rx 180 ry 0 rz -39.83 deg; joints [42.926, -59.873, 62.613, -0.858, 87.184, 42.964]
  MoveL 140 to (36.5, 248.56, 0) mm, rotated rx 180 ry 0 rz -39.83 deg; joints [42.916, -59.887, 62.634, -0.858, 87.177, 42.954]
  MoveL 141 to (36.36, 248.43, 0) mm, rotated rx 180 ry 0 rz -39.83 deg; joints [42.909, -59.897, 62.649, -0.858, 87.172, 42.948]
  MoveL 142 to (36.23, 248.3, 0) mm, rotated rx -180 ry 0 rz -39.83 deg; joints [42.902, -59.908, 62.665, -0.858, 87.167, 42.941]
  MoveL 143 to (36.12, 248.16, 0) mm, rotated rx 180 ry 0 rz -39.83 deg; joints [42.896, -59.919, 62.682, -0.858, 87.161, 42.935]
  MoveL 144 to (36.01, 248.01, 0) mm, rotated rx 180 ry 0 rz -39.83 deg; joints [42.891, -59.932, 62.701, -0.858, 87.155, 42.93]
  MoveL 145 to (35.94, 247.86, 0) mm, rotated rx 180 ry 0 rz -39.83 deg; joints [42.887, -59.945, 62.72, -0.858, 87.148, 42.926]
  MoveL 146 to (35.87, 247.7, 0) mm, rotated rx 180 ry 0 rz -39.83 deg; joints [42.883, -59.958, 62.74, -0.858, 87.142, 42.922]
  MoveL 147 to (35.82, 247.54, 0) mm, rotated rx 180 ry 0 rz -39.83 deg; joints [42.879, -59.972, 62.762, -0.858, 87.134, 42.919]
  MoveL 148 to (35.77, 247.38, 0) mm, rotated rx 180 ry 0 rz -39.83 deg; joints [42.876, -59.987, 62.783, -0.858, 87.127, 42.915]
  MoveL 149 to (35.77, 247.38, 0) mm, rotated rx 180 ry 0 rz -39.83 deg; joints [42.876, -59.987, 62.783, -0.858, 87.127, 42.915]
  MoveL 150 to (35.17, 247.41, 0) mm, rotated rx 180 ry 0 rz -39.83 deg; joints [42.85, -59.977, 62.768, -0.858, 87.132, 42.889]
  MoveL 151 to (34.58, 247.44, 0) mm, rotated rx 180 ry 0 rz -39.83 deg; joints [42.824, -59.967, 62.753, -0.858, 87.138, 42.863]
  MoveL 152 to (33.99, 247.46, 0) mm, rotated rx -180 ry 0 rz -39.83 deg; joints [42.797, -59.958, 62.739, -0.858, 87.143, 42.836]
  MoveL 153 to (33.4, 247.47, 0) mm, rotated rx 180 ry 0 rz -39.83 deg; joints [42.771, -59.951, 62.726, -0.858, 87.147, 42.81]
  MoveL 154 to (32.83, 247.47, 0) mm, rotated rx 180 ry 0 rz -39.83 deg; joints [42.745, -59.944, 62.715, -0.858, 87.151, 42.784]
  MoveL 155 to (32.27, 247.46, 0) mm, rotated rx 180 ry 0 rz -39.83 deg; joints [42.72, -59.938, 62.706, -0.858, 87.154, 42.759]
  MoveL 156 to (31.7, 247.44, 0) mm, rotated rx -180 ry 0 rz -39.83 deg; joints [42.694, -59.934, 62.698, -0.858, 87.157, 42.733]
  MoveL 157 to (31.13, 247.4, 0) mm, rotated rx 180 ry 0 rz -39.83 deg; joints [42.669, -59.93, 62.692, -0.858, 87.159, 42.707]
  MoveL 158 to (30.62, 247.37, 0) mm, rotated rx 180 ry 0 rz -39.83 deg; joints [42.646, -59.927, 62.687, -0.858, 87.161, 42.684]
  MoveL 159 to (30.11, 247.33, 0) mm, rotated rx 180 ry 0 rz -39.83 deg; joints [42.622, -59.925, 62.683, -0.858, 87.162, 42.661]
  MoveL 160 to (29.6, 247.27, 0) mm, rotated rx 180 ry 0 rz -39.83 deg; joints [42.599, -59.924, 62.68, -0.858, 87.163, 42.638]
  MoveL 161 to (29.09, 247.2, 0) mm, rotated rx 180 ry 0 rz -39.83 deg; joints [42.576, -59.924, 62.68, -0.858, 87.163, 42.615]
  MoveL 162 to (28.83, 247.16, 0) mm, rotated rx -180 ry 0 rz -39.83 deg; joints [42.564, -59.925, 62.681, -0.858, 87.163, 42.603]
  MoveL 163 to (28.57, 247.11, 0) mm, rotated rx 180 ry 0 rz -39.83 deg; joints [42.552, -59.926, 62.683, -0.858, 87.162, 42.591]
  MoveL 164 to (28.31, 247.06, 0) mm, rotated rx 180 ry 0 rz -39.83 deg; joints [42.54, -59.928, 62.685, -0.858, 87.162, 42.579]
  MoveL 165 to (28.05, 247, 0) mm, rotated rx 180 ry 0 rz -39.83 deg; joints [42.528, -59.93, 62.688, -0.858, 87.161, 42.567]
  MoveL 166 to (27.67, 246.91, 0) mm, rotated rx 180 ry 0 rz -39.83 deg; joints [42.511, -59.934, 62.693, -0.858, 87.159, 42.55]
  MoveL 167 to (27.3, 246.79, 0) mm, rotated rx 180 ry 0 rz -39.83 deg; joints [42.494, -59.94, 62.702, -0.858, 87.156, 42.532]
  MoveL 168 to (26.95, 246.65, 0) mm, rotated rx 180 ry 0 rz -39.83 deg; joints [42.477, -59.949, 62.715, -0.858, 87.152, 42.516]
  MoveL 169 to (26.62, 246.46, 0) mm, rotated rx -180 ry 0 rz -39.83 deg; joints [42.461, -59.962, 62.734, -0.858, 87.145, 42.5]
  MoveL 170 to (26.4, 246.3, 0) mm, rotated rx -180 ry 0 rz -39.83 deg; joints [42.45, -59.974, 62.752, -0.858, 87.139, 42.489]
  MoveL 171 to (26.2, 246.12, 0) mm, rotated rx 180 ry 0 rz -39.83 deg; joints [42.44, -59.988, 62.773, -0.858, 87.132, 42.479]
  MoveL 172 to (26, 245.92, 0) mm, rotated rx 180 ry 0 rz -39.83 deg; joints [42.43, -60.003, 62.796, -0.858, 87.125, 42.469]
  MoveL 173 to (25.82, 245.72, 0) mm, rotated rx 180 ry 0 rz -39.83 deg; joints [42.421, -60.02, 62.82, -0.858, 87.116, 42.46]
  MoveL 174 to (25.61, 245.46, 0) mm, rotated rx 180 ry 0 rz -39.83 deg; joints [42.41, -60.04, 62.851, -0.858, 87.106, 42.449]
  MoveL 175 to (25.4, 245.2, 0) mm, rotated rx 180 ry 0 rz -39.83 deg; joints [42.399, -60.062, 62.883, -0.858, 87.095, 42.438]
  MoveL 176 to (25.2, 244.93, 0) mm, rotated rx 180 ry 0 rz -39.83 deg; joints [42.388, -60.083, 62.915, -0.858, 87.084, 42.428]
  MoveL 177 to (25.01, 244.66, 0) mm, rotated rx 180 ry 0 rz -39.83 deg; joints [42.378, -60.105, 62.949, -0.858, 87.073, 42.418]
  MoveL 178 to (24.87, 244.46, 0) mm, rotated rx 180 ry 0 rz -39.83 deg; joints [42.371, -60.122, 62.974, -0.858, 87.065, 42.411]
  MoveL 179 to (24.73, 244.26, 0) mm, rotated rx 180 ry 0 rz -39.83 deg; joints [42.363, -60.139, 62.999, -0.858, 87.056, 42.403]
  MoveL 180 to (24.6, 244.05, 0) mm, rotated rx 180 ry 0 rz -39.83 deg; joints [42.356, -60.156, 63.024, -0.858, 87.048, 42.396]
  MoveL 181 to (24.46, 243.85, 0) mm, rotated rx 180 ry 0 rz -39.83 deg; joints [42.348, -60.173, 63.05, -0.858, 87.039, 42.389]
  MoveL 182 to (24.46, 243.85, 0) mm, rotated rx 180 ry 0 rz -39.83 deg; joints [42.348, -60.173, 63.05, -0.858, 87.039, 42.389]
  MoveL 183 to (24.33, 243.86, 0) mm, rotated rx 180 ry 0 rz -39.83 deg; joints [42.343, -60.17, 63.045, -0.858, 87.041, 42.383]
  MoveL 184 to (24.21, 243.88, 0) mm, rotated rx 180 ry 0 rz -39.83 deg; joints [42.337, -60.167, 63.04, -0.858, 87.042, 42.377]
  MoveL 185 to (24.08, 243.9, 0) mm, rotated rx 180 ry 0 rz -39.83 deg; joints [42.331, -60.164, 63.035, -0.858, 87.044, 42.372]
  MoveL 186 to (23.95, 243.91, 0) mm, rotated rx 180 ry 0 rz -39.83 deg; joints [42.326, -60.161, 63.03, -0.858, 87.046, 42.366]
  MoveL 187 to (23.7, 243.95, 0) mm, rotated rx 180 ry 0 rz -39.83 deg; joints [42.315, -60.154, 63.02, -0.858, 87.049, 42.355]
  MoveL 188 to (23.45, 243.99, 0) mm, rotated rx 180 ry 0 rz -39.83 deg; joints [42.304, -60.148, 63.01, -0.858, 87.053, 42.344]
  MoveL 189 to (23.2, 244.02, 0) mm, rotated rx 180 ry 0 rz -39.83 deg; joints [42.293, -60.141, 63, -0.858, 87.056, 42.333]
  MoveL 190 to (22.95, 244.05, 0) mm, rotated rx 180 ry 0 rz -39.83 deg; joints [42.282, -60.136, 62.991, -0.858, 87.059, 42.322]
  MoveL 191 to (22.52, 244.09, 0) mm, rotated rx 180 ry 0 rz -39.83 deg; joints [42.263, -60.127, 62.978, -0.857, 87.064, 42.303]
  MoveL 192 to (22.09, 244.1, 0) mm, rotated rx -180 ry 0 rz -39.83 deg; joints [42.243, -60.12, 62.967, -0.857, 87.067, 42.283]
  MoveL 193 to (21.65, 244.1, 0) mm, rotated rx 180 ry 0 rz -39.83 deg; joints [42.224, -60.115, 62.959, -0.857, 87.07, 42.264]
  MoveL 194 to (21.22, 244.09, 0) mm, rotated rx 180 ry 0 rz -39.83 deg; joints [42.205, -60.111, 62.952, -0.857, 87.073, 42.245]
  MoveL 195 to (20.89, 244.07, 0) mm, rotated rx 180 ry 0 rz -39.83 deg; joints [42.19, -60.108, 62.947, -0.857, 87.074, 42.23]
  MoveL 196 to (20.56, 244.04, 0) mm, rotated rx 180 ry 0 rz -39.83 deg; joints [42.175, -60.106, 62.944, -0.857, 87.075, 42.215]
  MoveL 197 to (20.23, 244.01, 0) mm, rotated rx 180 ry 0 rz -39.83 deg; joints [42.16, -60.106, 62.943, -0.857, 87.076, 42.2]
  MoveL 198 to (19.91, 243.95, 0) mm, rotated rx 180 ry 0 rz -39.83 deg; joints [42.145, -60.107, 62.944, -0.857, 87.076, 42.185]
  MoveL 199 to (19.58, 243.87, 0) mm, rotated rx 180 ry 0 rz -39.83 deg; joints [42.13, -60.11, 62.948, -0.857, 87.074, 42.17]
  MoveL 200 to (19.26, 243.77, 0) mm, rotated rx 180 ry 0 rz -39.83 deg; joints [42.115, -60.115, 62.956, -0.857, 87.072, 42.155]
  MoveL 201 to (18.94, 243.64, 0) mm, rotated rx -180 ry 0 rz -39.83 deg; joints [42.1, -60.122, 62.966, -0.857, 87.068, 42.14]
  MoveL 202 to (18.63, 243.5, 0) mm, rotated rx -180 ry 0 rz -39.83 deg; joints [42.085, -60.131, 62.979, -0.857, 87.064, 42.125]
  MoveL 203 to (18.36, 243.35, 0) mm, rotated rx -180 ry 0 rz -39.83 deg; joints [42.072, -60.141, 62.994, -0.857, 87.059, 42.112]
  MoveL 204 to (18.09, 243.19, 0) mm, rotated rx -180 ry 0 rz -39.83 deg; joints [42.059, -60.153, 63.011, -0.857, 87.053, 42.099]
  MoveL 205 to (17.84, 243.01, 0) mm, rotated rx 180 ry 0 rz -39.83 deg; joints [42.046, -60.166, 63.031, -0.857, 87.047, 42.087]
  MoveL 206 to (17.6, 242.81, 0) mm, rotated rx -180 ry 0 rz -39.83 deg; joints [42.034, -60.181, 63.052, -0.857, 87.04, 42.075]
  MoveL 207 to (17.25, 242.48, 0) mm, rotated rx 180 ry 0 rz -39.83 deg; joints [42.016, -60.206, 63.09, -0.857, 87.027, 42.057]
  MoveL 208 to (16.93, 242.12, 0) mm, rotated rx 180 ry 0 rz -39.83 deg; joints [42, -60.235, 63.133, -0.857, 87.013, 42.04]
  MoveL 209 to (16.63, 241.73, 0) mm, rotated rx 180 ry 0 rz -39.83 deg; joints [41.984, -60.266, 63.179, -0.857, 86.997, 42.025]
  MoveL 210 to (16.36, 241.33, 0) mm, rotated rx -180 ry 0 rz -39.83 deg; joints [41.969, -60.299, 63.229, -0.857, 86.98, 42.01]
  MoveL 211 to (16.18, 241.03, 0) mm, rotated rx 180 ry 0 rz -39.83 deg; joints [41.959, -60.324, 63.266, -0.857, 86.968, 42]
  MoveL 212 to (16.01, 240.73, 0) mm, rotated rx 180 ry 0 rz -39.83 deg; joints [41.95, -60.349, 63.304, -0.857, 86.955, 41.991]
  MoveL 213 to (15.87, 240.41, 0) mm, rotated rx 180 ry 0 rz -39.83 deg; joints [41.941, -60.376, 63.344, -0.857, 86.942, 41.983]
  MoveL 214 to (15.77, 240.09, 0) mm, rotated rx 180 ry 0 rz -39.83 deg; joints [41.935, -60.404, 63.386, -0.857, 86.928, 41.977]
  MoveL 215 to (15.7, 239.71, 0) mm, rotated rx 180 ry 0 rz -39.83 deg; joints [41.929, -60.437, 63.436, -0.857, 86.911, 41.971]
  MoveL 216 to (15.67, 239.32, 0) mm, rotated rx 180 ry 0 rz -39.83 deg; joints [41.925, -60.472, 63.488, -0.857, 86.894, 41.968]
  MoveL 217 to (15.67, 238.93, 0) mm, rotated rx -180 ry 0 rz -39.83 deg; joints [41.922, -60.507, 63.541, -0.857, 86.876, 41.965]
  MoveL 218 to (15.67, 238.54, 0) mm, rotated rx 180 ry 0 rz -39.83 deg; joints [41.92, -60.543, 63.594, -0.857, 86.858, 41.963]
  MoveL 219 to (15.67, 238.21, 0) mm, rotated rx 180 ry 0 rz -39.83 deg; joints [41.918, -60.573, 63.639, -0.857, 86.843, 41.961]
  MoveL 220 to (15.67, 237.88, 0) mm, rotated rx 180 ry 0 rz -39.83 deg; joints [41.915, -60.602, 63.684, -0.857, 86.828, 41.959]
  MoveL 221 to (15.67, 237.55, 0) mm, rotated rx -180 ry 0 rz -39.83 deg; joints [41.913, -60.632, 63.728, -0.857, 86.813, 41.957]
  MoveL 222 to (15.68, 237.22, 0) mm, rotated rx 180 ry 0 rz -39.83 deg; joints [41.912, -60.662, 63.773, -0.857, 86.798, 41.956]
  MoveL 223 to (15.71, 236.9, 0) mm, rotated rx 180 ry 0 rz -39.83 deg; joints [41.911, -60.691, 63.817, -0.857, 86.784, 41.955]
  MoveL 224 to (15.75, 236.59, 0) mm, rotated rx 180 ry 0 rz -39.83 deg; joints [41.911, -60.72, 63.86, -0.857, 86.769, 41.955]
  MoveL 225 to (15.81, 236.27, 0) mm, rotated rx 180 ry 0 rz -39.83 deg; joints [41.912, -60.749, 63.904, -0.857, 86.755, 41.956]
  MoveL 226 to (15.9, 235.97, 0) mm, rotated rx 180 ry 0 rz -39.83 deg; joints [41.913, -60.778, 63.947, -0.857, 86.74, 41.958]
  MoveL 227 to (15.99, 235.71, 0) mm, rotated rx -180 ry 0 rz -39.83 deg; joints [41.916, -60.802, 63.984, -0.857, 86.728, 41.961]
  MoveL 228 to (16.11, 235.46, 0) mm, rotated rx 180 ry 0 rz -39.83 deg; joints [41.919, -60.826, 64.02, -0.857, 86.716, 41.965]
  MoveL 229 to (16.24, 235.22, 0) mm, rotated rx -180 ry 0 rz -39.83 deg; joints [41.924, -60.85, 64.055, -0.857, 86.704, 41.969]
  MoveL 230 to (16.38, 234.98, 0) mm, rotated rx -180 ry 0 rz -39.83 deg; joints [41.929, -60.873, 64.089, -0.857, 86.693, 41.974]
  MoveL 231 to (16.52, 234.79, 0) mm, rotated rx 180 ry 0 rz -39.83 deg; joints [41.934, -60.891, 64.118, -0.857, 86.684, 41.979]
  MoveL 232 to (16.66, 234.61, 0) mm, rotated rx 180 ry 0 rz -39.83 deg; joints [41.939, -60.91, 64.145, -0.857, 86.674, 41.985]
  MoveL 233 to (16.81, 234.43, 0) mm, rotated rx 180 ry 0 rz -39.83 deg; joints [41.944, -60.928, 64.173, -0.857, 86.665, 41.99]
  MoveL 234 to (16.96, 234.25, 0) mm, rotated rx 180 ry 0 rz -39.83 deg; joints [41.95, -60.946, 64.2, -0.857, 86.656, 41.996]
  MoveL 235 to (16.96, 234.25, 0) mm, rotated rx 180 ry 0 rz -39.83 deg; joints [41.95, -60.946, 64.2, -0.857, 86.656, 41.996]
  MoveL 236 to (16.86, 234.13, 0) mm, rotated rx 180 ry 0 rz -39.83 deg; joints [41.945, -60.955, 64.214, -0.857, 86.652, 41.991]
  MoveL 237 to (16.77, 234.02, 0) mm, rotated rx -180 ry 0 rz -39.83 deg; joints [41.94, -60.965, 64.227, -0.857, 86.647, 41.986]
  MoveL 238 to (16.67, 233.9, 0) mm, rotated rx 180 ry 0 rz -39.83 deg; joints [41.935, -60.974, 64.241, -0.857, 86.643, 41.981]
  MoveL 239 to (16.57, 233.78, 0) mm, rotated rx 180 ry 0 rz -39.83 deg; joints [41.93, -60.983, 64.255, -0.857, 86.638, 41.976]
  MoveL 240 to (16.38, 233.54, 0) mm, rotated rx -180 ry 0 rz -39.83 deg; joints [41.919, -61.002, 64.283, -0.857, 86.629, 41.966]
  MoveL 241 to (16.19, 233.3, 0) mm, rotated rx 180 ry 0 rz -39.83 deg; joints [41.909, -61.021, 64.311, -0.857, 86.619, 41.956]
  MoveL 242 to (16.01, 233.05, 0) mm, rotated rx 180 ry 0 rz -39.83 deg; joints [41.899, -61.041, 64.341, -0.857, 86.61, 41.946]
  MoveL 243 to (15.85, 232.8, 0) mm, rotated rx 180 ry 0 rz -39.83 deg; joints [41.89, -61.062, 64.372, -0.857, 86.599, 41.937]
  MoveL 244 to (15.67, 232.46, 0) mm, rotated rx 180 ry 0 rz -39.83 deg; joints [41.88, -61.09, 64.414, -0.857, 86.586, 41.927]
  MoveL 245 to (15.53, 232.1, 0) mm, rotated rx 180 ry 0 rz -39.83 deg; joints [41.872, -61.12, 64.458, -0.857, 86.571, 41.919]
  MoveL 246 to (15.42, 231.74, 0) mm, rotated rx 180 ry 0 rz -39.83 deg; joints [41.864, -61.152, 64.505, -0.857, 86.555, 41.912]
  MoveL 247 to (15.33, 231.36, 0) mm, rotated rx 180 ry 0 rz -39.83 deg; joints [41.858, -61.184, 64.553, -0.857, 86.54, 41.906]
  MoveL 248 to (15.27, 230.98, 0) mm, rotated rx 180 ry 0 rz -39.83 deg; joints [41.852, -61.218, 64.604, -0.857, 86.523, 41.9]
  MoveL 249 to (15.23, 230.59, 0) mm, rotated rx -180 ry 0 rz -39.83 deg; joints [41.848, -61.253, 64.655, -0.857, 86.506, 41.896]
  MoveL 250 to (15.21, 230.2, 0) mm, rotated rx -180 ry 0 rz -39.83 deg; joints [41.844, -61.287, 64.707, -0.857, 86.489, 41.893]
  MoveL 251 to (15.2, 229.8, 0) mm, rotated rx 180 ry 0 rz -39.83 deg; joints [41.842, -61.322, 64.759, -0.857, 86.472, 41.89]
  MoveL 252 to (15.22, 229.35, 0) mm, rotated rx -180 ry 0 rz -39.83 deg; joints [41.839, -61.363, 64.82, -0.857, 86.452, 41.888]
  MoveL 253 to (15.26, 228.89, 0) mm, rotated rx 180 ry 0 rz -39.83 deg; joints [41.838, -61.405, 64.882, -0.857, 86.431, 41.887]
  MoveL 254 to (15.32, 228.44, 0) mm, rotated rx 180 ry 0 rz -39.83 deg; joints [41.838, -61.446, 64.943, -0.857, 86.411, 41.887]
  MoveL 255 to (15.4, 227.99, 0) mm, rotated rx 180 ry 0 rz -39.83 deg; joints [41.838, -61.487, 65.005, -0.857, 86.391, 41.888]
  MoveL 256 to (15.49, 227.59, 0) mm, rotated rx -180 ry 0 rz -39.83 deg; joints [41.84, -61.524, 65.059, -0.857, 86.373, 41.89]
  MoveL 257 to (15.6, 227.2, 0) mm, rotated rx 180 ry 0 rz -39.83 deg; joints [41.842, -61.56, 65.113, -0.857, 86.356, 41.893]
  MoveL 258 to (15.73, 226.82, 0) mm, rotated rx -180 ry 0 rz -39.83 deg; joints [41.846, -61.596, 65.166, -0.857, 86.338, 41.897]
  MoveL 259 to (15.89, 226.45, 0) mm, rotated rx 180 ry 0 rz -39.83 deg; joints [41.85, -61.631, 65.219, -0.857, 86.321, 41.901]
  MoveL 260 to (16.19, 225.86, 0) mm, rotated rx -180 ry 0 rz -39.83 deg; joints [41.86, -61.688, 65.303, -0.858, 86.293, 41.912]
  MoveL 261 to (16.54, 225.29, 0) mm, rotated rx -180 ry 0 rz -39.83 deg; joints [41.872, -61.743, 65.385, -0.858, 86.266, 41.924]
  MoveL 262 to (16.91, 224.74, 0) mm, rotated rx 180 ry 0 rz -39.83 deg; joints [41.885, -61.797, 65.466, -0.858, 86.24, 41.938]
  MoveL 263 to (17.3, 224.19, 0) mm, rotated rx 180 ry 0 rz -39.83 deg; joints [41.9, -61.85, 65.546, -0.858, 86.214, 41.952]
  MoveL 264 to (17.3, 224.19, 0) mm, rotated rx 180 ry 0 rz -39.83 deg; joints [41.9, -61.85, 65.546, -0.858, 86.214, 41.952]
  MoveL 265 to (17.15, 223.89, 0) mm, rotated rx 180 ry 0 rz -39.83 deg; joints [41.891, -61.875, 65.582, -0.858, 86.202, 41.944]
  MoveL 266 to (17.02, 223.59, 0) mm, rotated rx -180 ry 0 rz -39.83 deg; joints [41.883, -61.9, 65.618, -0.858, 86.19, 41.936]
  MoveL 267 to (16.91, 223.29, 0) mm, rotated rx -180 ry 0 rz -39.83 deg; joints [41.876, -61.925, 65.656, -0.858, 86.178, 41.929]
  MoveL 268 to (16.83, 222.98, 0) mm, rotated rx 180 ry 0 rz -39.83 deg; joints [41.87, -61.952, 65.696, -0.858, 86.165, 41.924]
  MoveL 269 to (16.81, 222.72, 0) mm, rotated rx 180 ry 0 rz -39.83 deg; joints [41.867, -61.975, 65.73, -0.858, 86.154, 41.921]
  MoveL 270 to (16.81, 222.45, 0) mm, rotated rx 180 ry 0 rz -39.83 deg; joints [41.866, -61.999, 65.764, -0.858, 86.143, 41.919]
  MoveL 271 to (16.82, 222.18, 0) mm, rotated rx -180 ry 0 rz -39.83 deg; joints [41.864, -62.023, 65.8, -0.858, 86.131, 41.918]
  MoveL 272 to (16.83, 221.91, 0) mm, rotated rx 180 ry 0 rz -39.83 deg; joints [41.863, -62.047, 65.835, -0.858, 86.12, 41.917]
  MoveL 273 to (16.85, 221.55, 0) mm, rotated rx 180 ry 0 rz -39.83 deg; joints [41.861, -62.079, 65.884, -0.858, 86.104, 41.916]
  MoveL 274 to (16.86, 221.19, 0) mm, rotated rx 180 ry 0 rz -39.83 deg; joints [41.86, -62.112, 65.931, -0.858, 86.089, 41.914]
  MoveL 275 to (16.88, 220.83, 0) mm, rotated rx 180 ry 0 rz -39.83 deg; joints [41.858, -62.144, 65.979, -0.858, 86.073, 41.913]
  MoveL 276 to (16.92, 220.47, 0) mm, rotated rx 180 ry 0 rz -39.83 deg; joints [41.857, -62.176, 66.027, -0.858, 86.058, 41.913]
  MoveL 277 to (16.97, 220.15, 0) mm, rotated rx 180 ry 0 rz -39.83 deg; joints [41.858, -62.205, 66.07, -0.858, 86.044, 41.913]
  MoveL 278 to (17.04, 219.83, 0) mm, rotated rx 180 ry 0 rz -39.83 deg; joints [41.859, -62.234, 66.112, -0.858, 86.03, 41.914]
  MoveL 279 to (17.13, 219.52, 0) mm, rotated rx 180 ry 0 rz -39.83 deg; joints [41.861, -62.263, 66.155, -0.858, 86.017, 41.917]
  MoveL 280 to (17.24, 219.21, 0) mm, rotated rx 180 ry 0 rz -39.83 deg; joints [41.864, -62.291, 66.197, -0.858, 86.003, 41.92]
  MoveL 281 to (17.45, 218.71, 0) mm, rotated rx 180 ry 0 rz -39.83 deg; joints [41.87, -62.339, 66.268, -0.858, 85.98, 41.926]
  MoveL 282 to (17.7, 218.22, 0) mm, rotated rx 180 ry 0 rz -39.83 deg; joints [41.878, -62.385, 66.336, -0.858, 85.958, 41.935]
  MoveL 283 to (17.99, 217.75, 0) mm, rotated rx -180 ry 0 rz -39.83 deg; joints [41.888, -62.43, 66.403, -0.858, 85.937, 41.945]
  MoveL 284 to (18.3, 217.3, 0) mm, rotated rx 180 ry 0 rz -39.83 deg; joints [41.9, -62.474, 66.468, -0.858, 85.916, 41.957]
  MoveL 285 to (18.69, 216.8, 0) mm, rotated rx 180 ry 0 rz -39.83 deg; joints [41.914, -62.523, 66.541, -0.858, 85.892, 41.972]
  MoveL 286 to (19.1, 216.32, 0) mm, rotated rx -180 ry 0 rz -39.83 deg; joints [41.93, -62.571, 66.611, -0.858, 85.87, 41.988]
  MoveL 287 to (19.53, 215.85, 0) mm, rotated rx 180 ry 0 rz -39.83 deg; joints [41.946, -62.618, 66.68, -0.858, 85.847, 42.004]
  MoveL 288 to (19.97, 215.39, 0) mm, rotated rx 180 ry 0 rz -39.83 deg; joints [41.963, -62.664, 66.749, -0.858, 85.825, 42.022]
  MoveL 289 to (19.97, 215.39, 0) mm, rotated rx 180 ry 0 rz -39.83 deg; joints [41.963, -62.664, 66.749, -0.858, 85.825, 42.022]
  MoveL 290 to (19.93, 215.07, 0) mm, rotated rx 180 ry 0 rz -39.83 deg; joints [41.959, -62.692, 66.79, -0.858, 85.812, 42.018]
  MoveL 291 to (19.89, 214.74, 0) mm, rotated rx -180 ry 0 rz -39.83 deg; joints [41.955, -62.72, 66.831, -0.858, 85.799, 42.014]
  MoveL 292 to (19.86, 214.42, 0) mm, rotated rx 180 ry 0 rz -39.83 deg; joints [41.952, -62.748, 66.873, -0.858, 85.786, 42.011]
  MoveL 293 to (19.84, 214.09, 0) mm, rotated rx 180 ry 0 rz -39.83 deg; joints [41.948, -62.777, 66.914, -0.858, 85.773, 42.008]
  MoveL 294 to (19.82, 213.74, 0) mm, rotated rx -180 ry 0 rz -39.83 deg; joints [41.945, -62.807, 66.959, -0.858, 85.758, 42.005]
  MoveL 295 to (19.81, 213.39, 0) mm, rotated rx 180 ry 0 rz -39.83 deg; joints [41.943, -62.838, 67.004, -0.858, 85.744, 42.002]
  MoveL 296 to (19.82, 213.04, 0) mm, rotated rx -180 ry 0 rz -39.83 deg; joints [41.941, -62.869, 67.05, -0.858, 85.729, 42.001]
  MoveL 297 to (19.84, 212.69, 0) mm, rotated rx -180 ry 0 rz -39.83 deg; joints [41.939, -62.9, 67.095, -0.858, 85.715, 41.999]
  MoveL 298 to (19.89, 212.26, 0) mm, rotated rx -180 ry 0 rz -39.83 deg; joints [41.939, -62.939, 67.152, -0.858, 85.697, 41.999]
  MoveL 299 to (19.96, 211.83, 0) mm, rotated rx 180 ry 0 rz -39.83 deg; joints [41.939, -62.978, 67.209, -0.858, 85.679, 42]
  MoveL 300 to (20.07, 211.4, 0) mm, rotated rx 180 ry 0 rz -39.83 deg; joints [41.941, -63.016, 67.265, -0.858, 85.661, 42.002]
  MoveL 301 to (20.2, 210.99, 0) mm, rotated rx 180 ry 0 rz -39.83 deg; joints [41.944, -63.054, 67.321, -0.858, 85.643, 42.006]
  MoveL 302 to (20.33, 210.65, 0) mm, rotated rx 180 ry 0 rz -39.83 deg; joints [41.948, -63.086, 67.367, -0.858, 85.628, 42.01]
  MoveL 303 to (20.49, 210.32, 0) mm, rotated rx 180 ry 0 rz -39.83 deg; joints [41.953, -63.116, 67.412, -0.858, 85.614, 42.015]
  MoveL 304 to (20.66, 210, 0) mm, rotated rx 180 ry 0 rz -39.83 deg; joints [41.959, -63.147, 67.457, -0.858, 85.6, 42.021]
  MoveL 305 to (20.84, 209.69, 0) mm, rotated rx -180 ry 0 rz -39.83 deg; joints [41.965, -63.176, 67.5, -0.858, 85.586, 42.027]
  MoveL 306 to (21.09, 209.3, 0) mm, rotated rx 180 ry 0 rz -39.83 deg; joints [41.974, -63.214, 67.556, -0.858, 85.569, 42.037]
  MoveL 307 to (21.37, 208.92, 0) mm, rotated rx 180 ry 0 rz -39.83 deg; joints [41.985, -63.251, 67.61, -0.859, 85.552, 42.047]
  MoveL 308 to (21.66, 208.55, 0) mm, rotated rx 180 ry 0 rz -39.83 deg; joints [41.996, -63.286, 67.662, -0.859, 85.535, 42.058]
  MoveL 309 to (21.97, 208.2, 0) mm, rotated rx 180 ry 0 rz -39.83 deg; joints [42.007, -63.321, 67.713, -0.859, 85.519, 42.071]
  MoveL 310 to (22.41, 207.74, 0) mm, rotated rx 180 ry 0 rz -39.83 deg; joints [42.025, -63.367, 67.781, -0.859, 85.497, 42.088]
  MoveL 311 to (22.88, 207.29, 0) mm, rotated rx -180 ry 0 rz -39.83 deg; joints [42.043, -63.412, 67.847, -0.859, 85.477, 42.107]
  MoveL 312 to (23.36, 206.86, 0) mm, rotated rx 180 ry 0 rz -39.83 deg; joints [42.063, -63.456, 67.911, -0.859, 85.456, 42.127]
  MoveL 313 to (23.85, 206.43, 0) mm, rotated rx 180 ry 0 rz -39.83 deg; joints [42.082, -63.499, 67.975, -0.859, 85.436, 42.147]
  MoveL 314 to (23.85, 206.43, 0) mm, rotated rx 180 ry 0 rz -39.83 deg; joints [42.082, -63.499, 67.975, -0.859, 85.436, 42.147]
  MoveL 315 to (23.81, 206.09, 0) mm, rotated rx 180 ry 0 rz -39.83 deg; joints [42.078, -63.529, 68.018, -0.859, 85.423, 42.143]
  MoveL 316 to (23.77, 205.74, 0) mm, rotated rx -180 ry 0 rz -39.83 deg; joints [42.074, -63.559, 68.061, -0.859, 85.409, 42.139]
  MoveL 317 to (23.75, 205.4, 0) mm, rotated rx -180 ry 0 rz -39.83 deg; joints [42.071, -63.588, 68.105, -0.859, 85.396, 42.136]
  MoveL 318 to (23.74, 205.05, 0) mm, rotated rx 180 ry 0 rz -39.83 deg; joints [42.068, -63.619, 68.149, -0.859, 85.382, 42.134]
  MoveL 319 to (23.76, 204.75, 0) mm, rotated rx -180 ry 0 rz -39.83 deg; joints [42.067, -63.645, 68.187, -0.859, 85.37, 42.133]
  MoveL 320 to (23.8, 204.46, 0) mm, rotated rx -180 ry 0 rz -39.83 deg; joints [42.067, -63.671, 68.225, -0.859, 85.358, 42.133]
  MoveL 321 to (23.85, 204.16, 0) mm, rotated rx 180 ry 0 rz -39.83 deg; joints [42.067, -63.698, 68.264, -0.859, 85.346, 42.133]
  MoveL 322 to (23.91, 203.86, 0) mm, rotated rx 180 ry 0 rz -39.83 deg; joints [42.069, -63.724, 68.303, -0.859, 85.334, 42.135]
  MoveL 323 to (24, 203.51, 0) mm, rotated rx -180 ry 0 rz -39.83 deg; joints [42.07, -63.756, 68.348, -0.859, 85.319, 42.137]
  MoveL 324 to (24.11, 203.17, 0) mm, rotated rx -180 ry 0 rz -39.83 deg; joints [42.073, -63.787, 68.394, -0.859, 85.305, 42.14]
  MoveL 325 to (24.24, 202.84, 0) mm, rotated rx 180 ry 0 rz -39.83 deg; joints [42.077, -63.818, 68.438, -0.859, 85.291, 42.144]
  MoveL 326 to (24.4, 202.53, 0) mm, rotated rx 180 ry 0 rz -39.83 deg; joints [42.082, -63.847, 68.481, -0.859, 85.278, 42.149]
  MoveL 327 to (24.68, 202.1, 0) mm, rotated rx 180 ry 0 rz -39.83 deg; joints [42.092, -63.888, 68.541, -0.859, 85.259, 42.16]
  MoveL 328 to (25.01, 201.7, 0) mm, rotated rx -180 ry 0 rz -39.83 deg; joints [42.105, -63.927, 68.598, -0.859, 85.242, 42.172]
  MoveL 329 to (25.37, 201.32, 0) mm, rotated rx 180 ry 0 rz -39.83 deg; joints [42.119, -63.964, 68.652, -0.859, 85.225, 42.187]
  MoveL 330 to (25.74, 200.95, 0) mm, rotated rx 180 ry 0 rz -39.83 deg; joints [42.134, -64, 68.705, -0.859, 85.208, 42.202]
  MoveL 331 to (26.17, 200.55, 0) mm, rotated rx 180 ry 0 rz -39.83 deg; joints [42.151, -64.041, 68.765, -0.859, 85.19, 42.22]
  MoveL 332 to (26.61, 200.15, 0) mm, rotated rx 180 ry 0 rz -39.83 deg; joints [42.169, -64.081, 68.823, -0.859, 85.172, 42.238]
  MoveL 333 to (27.05, 199.76, 0) mm, rotated rx 180 ry 0 rz -39.83 deg; joints [42.187, -64.12, 68.88, -0.859, 85.154, 42.256]
  MoveL 334 to (27.5, 199.38, 0) mm, rotated rx 180 ry 0 rz -39.83 deg; joints [42.206, -64.158, 68.936, -0.859, 85.136, 42.275]
  MoveL 335 to (28.16, 198.87, 0) mm, rotated rx 180 ry 0 rz -39.83 deg; joints [42.233, -64.211, 69.013, -0.859, 85.113, 42.302]
  MoveL 336 to (28.82, 198.37, 0) mm, rotated rx 180 ry 0 rz -39.83 deg; joints [42.26, -64.262, 69.088, -0.86, 85.089, 42.33]
  MoveL 337 to (29.5, 197.88, 0) mm, rotated rx 180 ry 0 rz -39.83 deg; joints [42.289, -64.312, 69.161, -0.86, 85.067, 42.359]
  MoveL 338 to (30.19, 197.4, 0) mm, rotated rx -180 ry 0 rz -39.83 deg; joints [42.318, -64.362, 69.234, -0.86, 85.044, 42.388]
  MoveL 339 to (30.19, 197.4, 0) mm, rotated rx -180 ry 0 rz -39.83 deg; joints [42.318, -64.362, 69.234, -0.86, 85.044, 42.388]
  MoveL 340 to (30.23, 197, 0) mm, rotated rx -180 ry 0 rz -39.83 deg; joints [42.317, -64.398, 69.285, -0.86, 85.028, 42.388]
  MoveL 341 to (30.29, 196.59, 0) mm, rotated rx 180 ry 0 rz -39.83 deg; joints [42.317, -64.434, 69.337, -0.86, 85.012, 42.388]
  MoveL 342 to (30.35, 196.19, 0) mm, rotated rx -180 ry 0 rz -39.83 deg; joints [42.318, -64.469, 69.389, -0.86, 84.997, 42.389]
  MoveL 343 to (30.44, 195.79, 0) mm, rotated rx 180 ry 0 rz -39.83 deg; joints [42.319, -64.505, 69.44, -0.86, 84.981, 42.391]
  MoveL 344 to (30.54, 195.46, 0) mm, rotated rx 180 ry 0 rz -39.83 deg; joints [42.321, -64.535, 69.483, -0.86, 84.968, 42.393]
  MoveL 345 to (30.65, 195.13, 0) mm, rotated rx 180 ry 0 rz -39.83 deg; joints [42.325, -64.565, 69.526, -0.86, 84.954, 42.397]
  MoveL 346 to (30.79, 194.81, 0) mm, rotated rx 180 ry 0 rz -39.83 deg; joints [42.329, -64.594, 69.569, -0.86, 84.941, 42.401]
  MoveL 347 to (30.95, 194.5, 0) mm, rotated rx 180 ry 0 rz -39.83 deg; joints [42.335, -64.623, 69.61, -0.86, 84.929, 42.407]
  MoveL 348 to (31.25, 194.03, 0) mm, rotated rx 180 ry 0 rz -39.83 deg; joints [42.346, -64.668, 69.675, -0.86, 84.909, 42.418]
  MoveL 349 to (31.6, 193.58, 0) mm, rotated rx 180 ry 0 rz -39.83 deg; joints [42.359, -64.71, 69.737, -0.86, 84.89, 42.432]
  MoveL 350 to (31.99, 193.17, 0) mm, rotated rx 180 ry 0 rz -39.83 deg; joints [42.375, -64.751, 69.795, -0.86, 84.872, 42.448]
  MoveL 351 to (32.41, 192.78, 0) mm, rotated rx -180 ry 0 rz -39.83 deg; joints [42.392, -64.789, 69.85, -0.86, 84.855, 42.465]
  MoveL 352 to (32.97, 192.34, 0) mm, rotated rx 180 ry 0 rz -39.83 deg; joints [42.415, -64.833, 69.915, -0.86, 84.835, 42.489]
  MoveL 353 to (33.55, 191.94, 0) mm, rotated rx 180 ry 0 rz -39.83 deg; joints [42.44, -64.875, 69.976, -0.86, 84.817, 42.513]
  MoveL 354 to (34.15, 191.57, 0) mm, rotated rx 180 ry 0 rz -39.83 deg; joints [42.465, -64.914, 70.032, -0.86, 84.8, 42.54]
  MoveL 355 to (34.77, 191.24, 0) mm, rotated rx 180 ry 0 rz -39.83 deg; joints [42.492, -64.95, 70.084, -0.86, 84.784, 42.567]
  MoveL 356 to (35.58, 190.85, 0) mm, rotated rx 180 ry 0 rz -39.83 deg; joints [42.528, -64.992, 70.146, -0.86, 84.765, 42.602]
  MoveL 357 to (36.4, 190.51, 0) mm, rotated rx 180 ry 0 rz -39.83 deg; joints [42.564, -65.032, 70.204, -0.86, 84.747, 42.639]
  MoveL 358 to (37.24, 190.18, 0) mm, rotated rx 180 ry 0 rz -39.83 deg; joints [42.601, -65.069, 70.258, -0.86, 84.731, 42.677]
  MoveL 359 to (38.08, 189.87, 0) mm, rotated rx -180 ry 0 rz -39.83 deg; joints [42.639, -65.105, 70.311, -0.861, 84.714, 42.714]
  MoveL 360 to (38.08, 189.87, 0) mm, rotated rx -180 ry 0 rz -39.83 deg; joints [42.639, -65.105, 70.311, -0.861, 84.714, 42.714]
  MoveL 361 to (38.06, 189.7, 0) mm, rotated rx -180 ry 0 rz -39.83 deg; joints [42.637, -65.12, 70.332, -0.861, 84.708, 42.712]
  MoveL 362 to (38.04, 189.53, 0) mm, rotated rx 180 ry 0 rz -39.83 deg; joints [42.635, -65.135, 70.353, -0.861, 84.702, 42.711]
  MoveL 363 to (38.03, 189.35, 0) mm, rotated rx 180 ry 0 rz -39.83 deg; joints [42.634, -65.149, 70.374, -0.861, 84.696, 42.709]
  MoveL 364 to (38.04, 189.18, 0) mm, rotated rx 180 ry 0 rz -39.83 deg; joints [42.633, -65.164, 70.395, -0.861, 84.689, 42.709]
  MoveL 365 to (38.06, 189, 0) mm, rotated rx 180 ry 0 rz -39.83 deg; joints [42.633, -65.18, 70.418, -0.861, 84.682, 42.709]
  MoveL 366 to (38.11, 188.82, 0) mm, rotated rx 180 ry 0 rz -39.83 deg; joints [42.634, -65.196, 70.441, -0.861, 84.675, 42.71]
  MoveL 367 to (38.16, 188.65, 0) mm, rotated rx 180 ry 0 rz -39.83 deg; joints [42.635, -65.212, 70.464, -0.861, 84.669, 42.711]
  MoveL 368 to (38.22, 188.47, 0) mm, rotated rx 180 ry 0 rz -39.83 deg; joints [42.637, -65.228, 70.486, -0.861, 84.662, 42.713]
  MoveL 369 to (38.37, 188.14, 0) mm, rotated rx 180 ry 0 rz -39.83 deg; joints [42.642, -65.258, 70.53, -0.861, 84.649, 42.718]
  MoveL 370 to (38.53, 187.81, 0) mm, rotated rx 180 ry 0 rz -39.83 deg; joints [42.647, -65.288, 70.573, -0.861, 84.636, 42.724]
  MoveL 371 to (38.71, 187.5, 0) mm, rotated rx 180 ry 0 rz -39.83 deg; joints [42.654, -65.317, 70.615, -0.861, 84.623, 42.731]
  MoveL 372 to (38.91, 187.19, 0) mm, rotated rx 180 ry 0 rz -39.83 deg; joints [42.661, -65.346, 70.656, -0.861, 84.611, 42.738]
  MoveL 373 to (39.19, 186.81, 0) mm, rotated rx 180 ry 0 rz -39.83 deg; joints [42.672, -65.382, 70.708, -0.861, 84.595, 42.75]
  MoveL 374 to (39.5, 186.45, 0) mm, rotated rx 180 ry 0 rz -39.83 deg; joints [42.685, -65.416, 70.757, -0.861, 84.58, 42.762]
  MoveL 375 to (39.84, 186.12, 0) mm, rotated rx -180 ry 0 rz -39.83 deg; joints [42.698, -65.448, 70.803, -0.861, 84.566, 42.776]
  MoveL 376 to (40.21, 185.83, 0) mm, rotated rx -180 ry 0 rz -39.83 deg; joints [42.714, -65.477, 70.845, -0.861, 84.554, 42.792]
  MoveL 377 to (40.64, 185.57, 0) mm, rotated rx -180 ry 0 rz -39.83 deg; joints [42.733, -65.505, 70.885, -0.861, 84.542, 42.811]
  MoveL 378 to (41.11, 185.35, 0) mm, rotated rx -180 ry 0 rz -39.83 deg; joints [42.753, -65.529, 70.919, -0.861, 84.531, 42.832]
  MoveL 379 to (41.59, 185.16, 0) mm, rotated rx -180 ry 0 rz -39.83 deg; joints [42.775, -65.551, 70.951, -0.861, 84.522, 42.853]
  MoveL 380 to (42.07, 184.97, 0) mm, rotated rx 180 ry 0 rz -39.83 deg; joints [42.797, -65.572, 70.982, -0.861, 84.513, 42.875]
  MoveL 381 to (42.74, 184.71, 0) mm, rotated rx 180 ry 0 rz -39.83 deg; joints [42.827, -65.602, 71.026, -0.861, 84.5, 42.905]
  MoveL 382 to (43.42, 184.45, 0) mm, rotated rx 180 ry 0 rz -39.83 deg; joints [42.857, -65.631, 71.068, -0.861, 84.487, 42.936]
  MoveL 383 to (44.1, 184.23, 0) mm, rotated rx 180 ry 0 rz -39.83 deg; joints [42.888, -65.658, 71.107, -0.861, 84.475, 42.967]
  MoveL 384 to (44.8, 184.05, 0) mm, rotated rx 180 ry 0 rz -39.83 deg; joints [42.92, -65.681, 71.141, -0.861, 84.465, 42.999]
  MoveL 385 to (45.15, 183.98, 0) mm, rotated rx 180 ry 0 rz -39.83 deg; joints [42.936, -65.69, 71.154, -0.861, 84.461, 43.015]
  MoveL 386 to (45.49, 183.91, 0) mm, rotated rx 180 ry 0 rz -39.83 deg; joints [42.951, -65.7, 71.169, -0.861, 84.456, 43.031]
  MoveL 387 to (45.82, 183.82, 0) mm, rotated rx 180 ry 0 rz -39.83 deg; joints [42.966, -65.712, 71.186, -0.861, 84.451, 43.046]
  MoveL 388 to (46.12, 183.68, 0) mm, rotated rx 180 ry 0 rz -39.83 deg; joints [42.98, -65.727, 71.208, -0.861, 84.445, 43.06]
  MoveL 389 to (46.28, 183.58, 0) mm, rotated rx -180 ry 0 rz -39.83 deg; joints [42.987, -65.737, 71.222, -0.861, 84.44, 43.066]
  MoveL 390 to (46.42, 183.47, 0) mm, rotated rx 180 ry 0 rz -39.83 deg; joints [42.993, -65.748, 71.239, -0.861, 84.435, 43.073]
  MoveL 391 to (46.57, 183.34, 0) mm, rotated rx -180 ry 0 rz -39.83 deg; joints [42.999, -65.76, 71.256, -0.861, 84.43, 43.079]
  MoveL 392 to (46.7, 183.22, 0) mm, rotated rx 180 ry 0 rz -39.83 deg; joints [43.005, -65.773, 71.274, -0.861, 84.425, 43.085]
  Establecer velocidad (1000.0 mm/s)
  MoveL 393 to (46.7, 183.22, 0) mm, rotated rx 180 ry 0 rz -39.83 deg; joints [43.005, -65.773, 71.274, -0.861, 84.425, 43.085]
  MoveL 394 to (46.7, 183.22, 20) mm, rotated rx 180 ry 0 rz -39.83 deg; joints [43.019, -66.01, 69.886, -0.859, 86.049, 43.074]

